(* CoDeSys 2.3.9.42 project: CFC,LAD,ST_81.pro *)

(* POU PLC_PRG, SFC *)
PROGRAM PLC_PRG
VAR
END_VAR
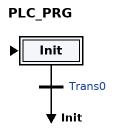
INITIAL_STEP Init:
END_STEP
TRANSITION FROM Init TO Init := Trans0;
END_TRANSITION
END_PROGRAM

(* POU CFC, CFC *)
PROGRAM CFC
VAR
	Y3: BOOL;
	Y2: BOOL;
	Y1: BOOL;
	X1: BOOL;
	X2: BOOL;
	X3: BOOL;
	X4: BOOL;
	X5: BOOL;
END_VAR
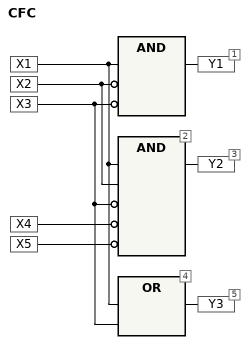
_CFC_ (* Continuous Function Chart, elements in execution order *)
#0 AND(X1, NOT X2, NOT X3)
#1 Y1 <= #0
#2 AND(X1, X2, NOT X3, NOT X4, NOT X5)
#3 Y2 <= #2
#4 OR(X1, X3)
#5 Y3 <= #4
_END_CFC_
(* the same logic as Structured Text *)
Y1 := X1 AND NOT X2 AND NOT X3;
Y2 := X1 AND X2 AND NOT X3 AND NOT X4 AND NOT X5;
Y3 := X1 OR X3;
END_PROGRAM

(* POU LAD, LD *)
PROGRAM LAD
VAR
	X1: BOOL;
	X2: BOOL;
	X3: BOOL;
	Y1: BOOL;
	Y3: BOOL;
	Y2: BOOL;
	X4: BOOL;
	X5: BOOL;
END_VAR
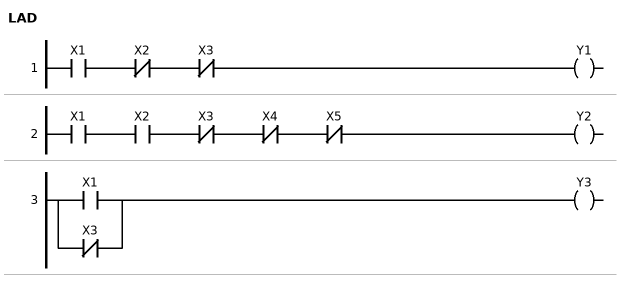
_LD_ (* Ladder Diagram *)
NETWORK 1
	[X1] - [/X2] - [/X3] --- (Y1)
NETWORK 2
	[X1] - [X2] - [/X3] - [/X4] - [/X5] --- (Y2)
NETWORK 3
	{ [X1] | [/X3] } --- (Y3)
_END_LD_
(* the same logic as Structured Text *)
(* Network 1 *)
Y1 := X1 AND NOT X2 AND NOT X3;
(* Network 2 *)
Y2 := X1 AND X2 AND NOT X3 AND NOT X4 AND NOT X5;
(* Network 3 *)
Y3 := X1 OR NOT X3;
END_PROGRAM

(* POU Structuret_text, ST *)
PROGRAM Structuret_text
VAR
	X1: BOOL;
	X2: BOOL;
	X3: BOOL;
	Y1: BOOL;
	X4: BOOL;
	X5: BOOL;
	Y2: BOOL;
	Y3: BOOL;
END_VAR
IF X1 AND (NOT X2) AND (NOT X3)
THEN
Y1 := TRUE;
ELSE
Y1:=FALSE;
END_IF

IF X1 AND X2 AND (NOT X3) AND (NOT X4) AND (NOT X5)
THEN
Y2:=TRUE;
ELSE
Y2:=FALSE;
END_IF

IF X1 OR (NOT X3)
THEN
Y3:=TRUE;
ELSE
Y3:=FALSE;
END_IF
END_PROGRAM
